(* IEC 61131-3 sources: verifaps-lib/geteta/examples, 1 file *)

(* ---- steps.st ---- *)
PROGRAM steps

VAR_OUTPUT o : INT := 0; END_VAR

o := o + 1;

END_PROGRAM
